// Mitsubishi GX Works2 project: 2023-06-20 #2 생산자동화기능사 20번   PLC: Q03UDV
// 생산자동화기능사

// global labels: Global1
VAR_GLOBAL
  PB1 AT X0 : BOOL;
  PB2 AT X1 : BOOL;
  정지 AT X2 : BOOL;
  공급후진 AT X3 : BOOL;
  공급전진 AT X4 : BOOL;
  가공후진 AT X5 : BOOL;
  가공전진 AT X6 : BOOL;
  송출후진 AT X7 : BOOL;
  송출전진 AT X8 : BOOL;
  배출후진 AT X9 : BOOL;
  배출전진 AT X0A : BOOL;
  매거진 AT X0B : BOOL;
  금속센서 AT X0F : BOOL;
  PB3 AT X10 : BOOL;
  적색 AT Y20 : BOOL;
  황색 AT Y21 : BOOL;
  녹색 AT Y22 : BOOL;
  공급1 AT Y23 : BOOL;
  공급2 AT Y24 : BOOL;
  가공 AT Y25 : BOOL;
  드릴 AT Y26 : BOOL;
  송출 AT Y27 : BOOL;
  배출 AT Y28 : BOOL;
  컨베이어 AT Y29 : BOOL;
END_VAR

PROGRAM 테스트동작
VAR
  PHASE : INT;
END_VAR
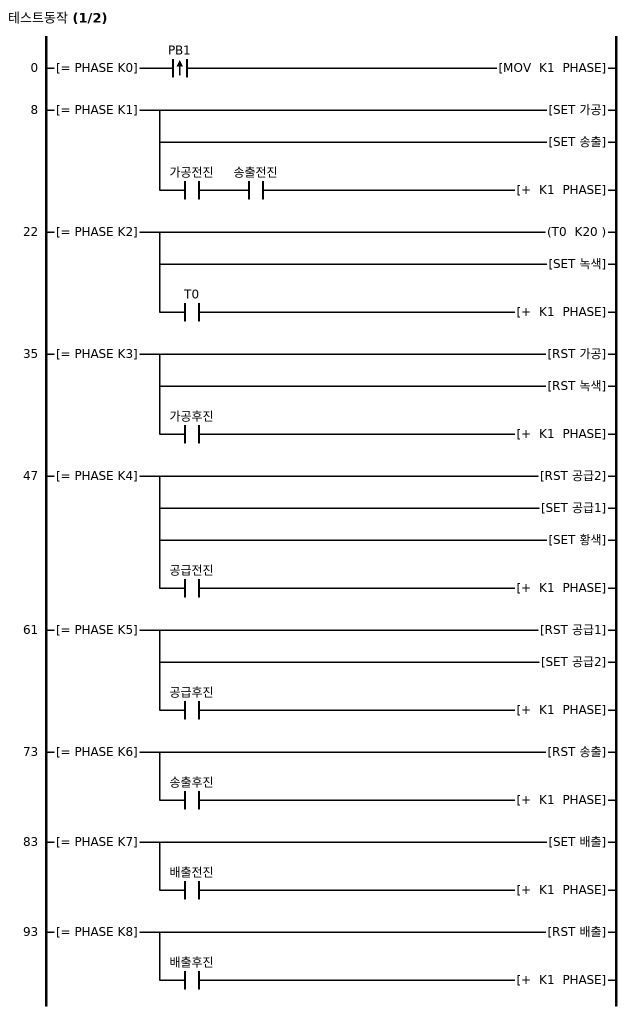
0     LD=     PHASE K0
      ANDP    PB1
      MOV     K1 PHASE
8     LD=     PHASE K1
      SET     가공
      SET     송출
      AND     가공전진
      AND     송출전진
      +       K1 PHASE
22    LD=     PHASE K2
      OUT     T0 K20
      SET     녹색
      AND     T0
      +       K1 PHASE
35    LD=     PHASE K3
      RST     가공
      RST     녹색
      AND     가공후진
      +       K1 PHASE
47    LD=     PHASE K4
      RST     공급2
      SET     공급1
      SET     황색
      AND     공급전진
      +       K1 PHASE
61    LD=     PHASE K5
      RST     공급1
      SET     공급2
      AND     공급후진
      +       K1 PHASE
73    LD=     PHASE K6
      RST     송출
      AND     송출후진
      +       K1 PHASE
83    LD=     PHASE K7
      SET     배출
      AND     배출전진
      +       K1 PHASE
93    LD=     PHASE K8
      RST     배출
      AND     배출후진
      +       K1 PHASE
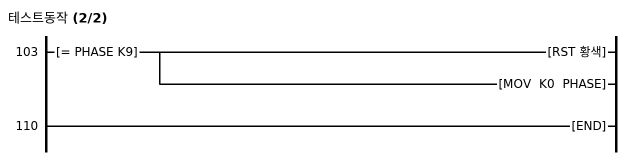
103   LD=     PHASE K9
      RST     황색
      MOV     K0 PHASE
110   END
END_PROGRAM

PROGRAM 생산자동화기능사
VAR
  PHASE : INT;
  MODE : INT;
END_VAR
VAR CONSTANT
  단속 : INT;
  연속 : INT := 1;
END_VAR
VAR
  BLINK : ARRAY [0..11] OF BOOL;
  METAL : INT;
END_VAR
VAR CONSTANT
  금속 : INT := 1;
  비금속 : INT := 2;
END_VAR
VAR
  LOOP : ARRAY [0..0] OF INT;
  EMG : INT;
END_VAR
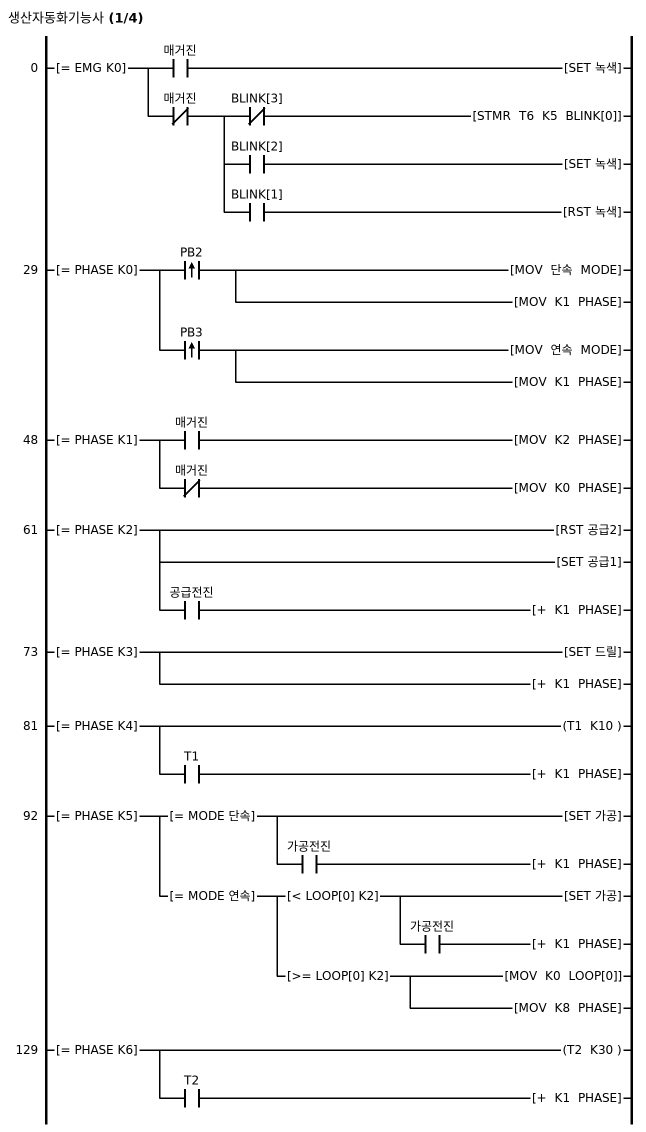
0     LD=     EMG K0
      MPS
      AND     매거진
      SET     녹색
      MPP
      ANI     매거진
      MPS
      ANI     BLINK[3]
      STMR    T6 K5 BLINK[0]
      MRD
      AND     BLINK[2]
      SET     녹색
      MPP
      AND     BLINK[1]
      RST     녹색
29    LD=     PHASE K0
      MPS
      ANDP    PB2
      MOV     단속 MODE
      MOV     K1 PHASE
      MPP
      ANDP    PB3
      MOV     연속 MODE
      MOV     K1 PHASE
48    LD=     PHASE K1
      MPS
      AND     매거진
      MOV     K2 PHASE
      MPP
      ANI     매거진
      MOV     K0 PHASE
61    LD=     PHASE K2
      RST     공급2
      SET     공급1
      AND     공급전진
      +       K1 PHASE
73    LD=     PHASE K3
      SET     드릴
      +       K1 PHASE
81    LD=     PHASE K4
      OUT     T1 K10
      AND     T1
      +       K1 PHASE
92    LD=     PHASE K5
      MPS
      AND=    MODE 단속
      SET     가공
      AND     가공전진
      +       K1 PHASE
      MPP
      AND=    MODE 연속
      MPS
      AND<    LOOP[0] K2
      SET     가공
      AND     가공전진
      +       K1 PHASE
      MPP
      AND>=   LOOP[0] K2
      MOV     K0 LOOP[0]
      MOV     K8 PHASE
129   LD=     PHASE K6
      OUT     T2 K30
      AND     T2
      +       K1 PHASE
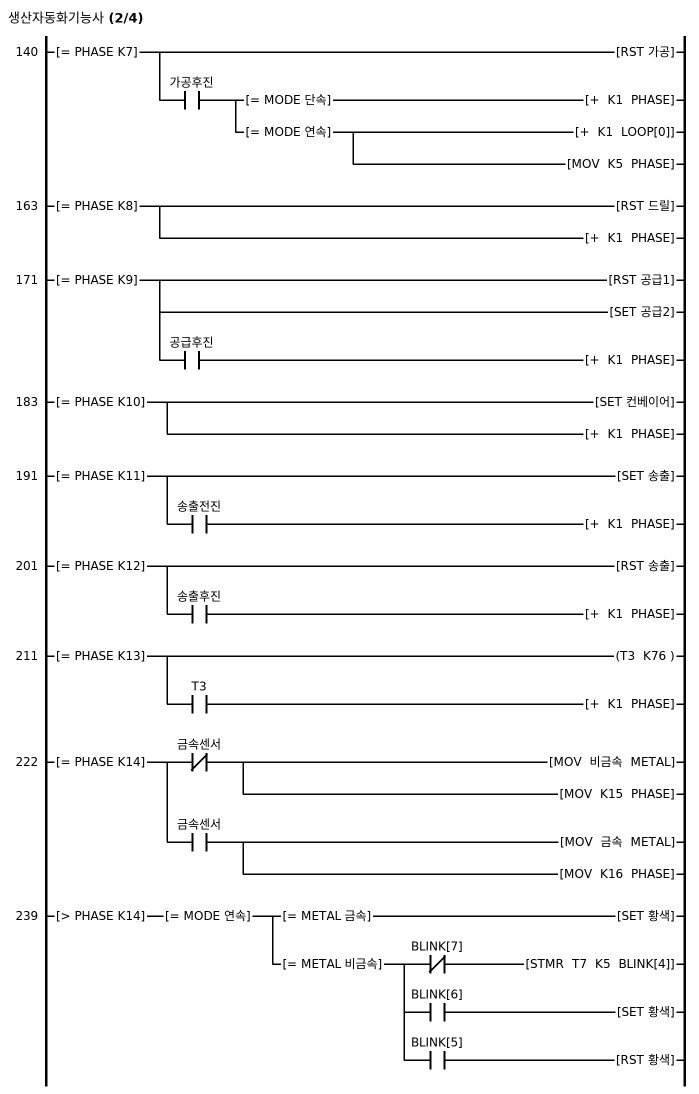
140   LD=     PHASE K7
      RST     가공
      AND     가공후진
      MPS
      AND=    MODE 단속
      +       K1 PHASE
      MPP
      AND=    MODE 연속
      +       K1 LOOP[0]
      MOV     K5 PHASE
163   LD=     PHASE K8
      RST     드릴
      +       K1 PHASE
171   LD=     PHASE K9
      RST     공급1
      SET     공급2
      AND     공급후진
      +       K1 PHASE
183   LD=     PHASE K10
      SET     컨베이어
      +       K1 PHASE
191   LD=     PHASE K11
      SET     송출
      AND     송출전진
      +       K1 PHASE
201   LD=     PHASE K12
      RST     송출
      AND     송출후진
      +       K1 PHASE
211   LD=     PHASE K13
      OUT     T3 K76
      AND     T3
      +       K1 PHASE
222   LD=     PHASE K14
      MPS
      ANI     금속센서
      MOV     비금속 METAL
      MOV     K15 PHASE
      MPP
      AND     금속센서
      MOV     금속 METAL
      MOV     K16 PHASE
239   LD>     PHASE K14
      AND=    MODE 연속
      MPS
      AND=    METAL 금속
      SET     황색
      MPP
      AND=    METAL 비금속
      MPS
      ANI     BLINK[7]
      STMR    T7 K5 BLINK[4]
      MRD
      AND     BLINK[6]
      SET     황색
      MPP
      AND     BLINK[5]
      RST     황색
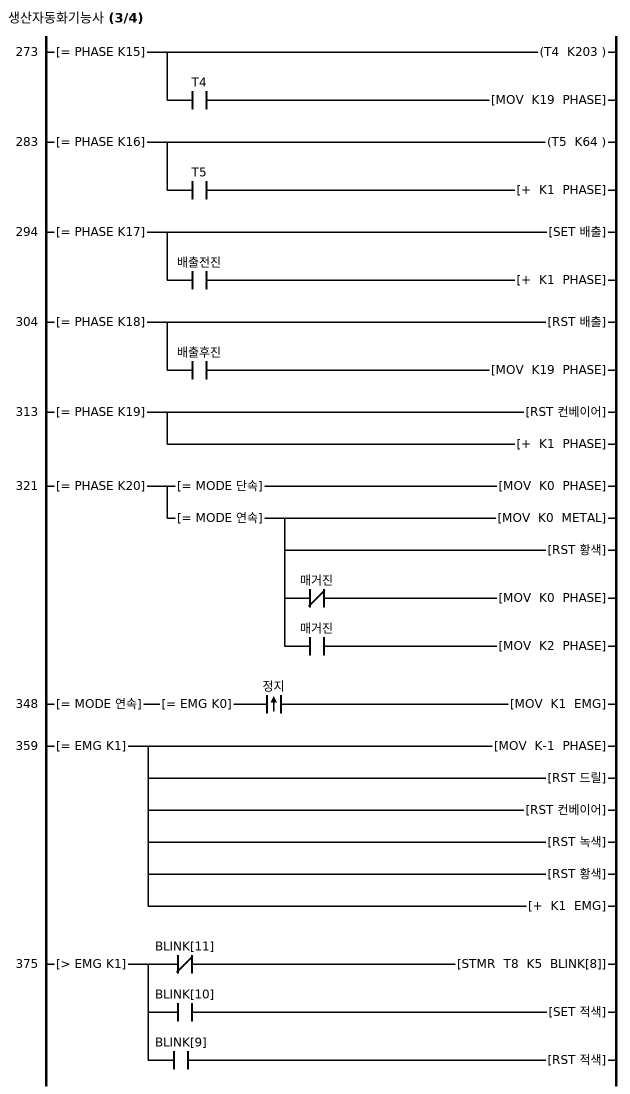
273   LD=     PHASE K15
      OUT     T4 K203
      AND     T4
      MOV     K19 PHASE
283   LD=     PHASE K16
      OUT     T5 K64
      AND     T5
      +       K1 PHASE
294   LD=     PHASE K17
      SET     배출
      AND     배출전진
      +       K1 PHASE
304   LD=     PHASE K18
      RST     배출
      AND     배출후진
      MOV     K19 PHASE
313   LD=     PHASE K19
      RST     컨베이어
      +       K1 PHASE
321   LD=     PHASE K20
      MPS
      AND=    MODE 단속
      MOV     K0 PHASE
      MPP
      AND=    MODE 연속
      MOV     K0 METAL
      RST     황색
      MPS
      ANI     매거진
      MOV     K0 PHASE
      MPP
      AND     매거진
      MOV     K2 PHASE
348   LD=     MODE 연속
      AND=    EMG K0
      ANDP    정지
      MOV     K1 EMG
359   LD=     EMG K1
      MOV     K-1 PHASE
      RST     드릴
      RST     컨베이어
      RST     녹색
      RST     황색
      +       K1 EMG
375   LD>     EMG K1
      MPS
      ANI     BLINK[11]
      STMR    T8 K5 BLINK[8]
      MRD
      AND     BLINK[10]
      SET     적색
      MPP
      AND     BLINK[9]
      RST     적색
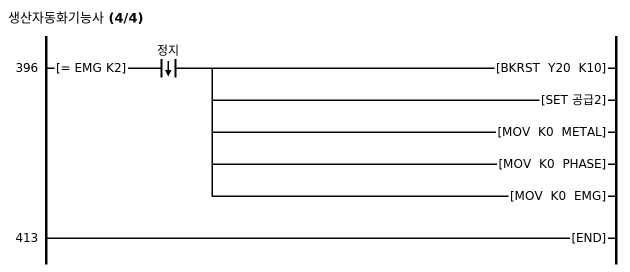
396   LD=     EMG K2
      ANDF    정지
      BKRST   Y20 K10
      SET     공급2
      MOV     K0 METAL
      MOV     K0 PHASE
      MOV     K0 EMG
413   END
END_PROGRAM
